FUNCTION_BLOCK FB_Food
VAR_OUTPUT
	stFood 				: ST_Food;
END_VAR
VAR
	randomColumnNumGenerator :	DRAND;
	randomRowNumGenerator 	:	DRAND;
	iRandColumn				:	INT;
 	iRandRow				:	INT;
END_VAR

randomColumnNumGenerator(Seed:= iRandColumn+10);
randomRowNumGenerator(Seed:= iRandRow);

iRandColumn := LREAL_TO_INT(randomColumnNumGenerator.Num * 9);
iRandRow 	:= LREAL_TO_INT(randomRowNumGenerator.Num * 9);

METHOD M_Generate : BOOL;
VAR_INPUT
	
END_VAR
M_Generate := FALSE;
	stFood.stFoodCoordinate.iColumnCoordinate := iRandColumn; 
	stFood.stFoodCoordinate.iRowCoordinate := iRandRow; 
M_Generate := TRUE;
END_METHOD

END_FUNCTION_BLOCK

(* stored: Version 1.1.0.1, ProductVersion 3.1.4024.4
   POU FB_Food: Id {5a554aa6-ff02-47a3-af06-484f1ba4dfb6}, SpecialFunc None
   Method M_Generate: Id {cafbc78c-a1d5-4f15-8b6b-3c5dbd0bab40} *)
